(* Specifies the operating mode of a PID controller. *)
{attribute 'qualified_only'}
{attribute 'strict'}
{attribute 'to_string'}
TYPE E_PIDMode :
(
	// Output tracks Setpoint directly through the output clamp.
	Auto 	:= 0,
	// Output is computed from Setpoint and Feedback using the PID algorithm.
	Manual	:= 1
)BYTE;
END_TYPE

(* stored: Version 1.1.0.1, ProductVersion 3.1.4024.15
   EnumerationTextList E_PIDMode: Id {ad840b95-c69a-0b49-1cff-63e9d69bb985} *)
